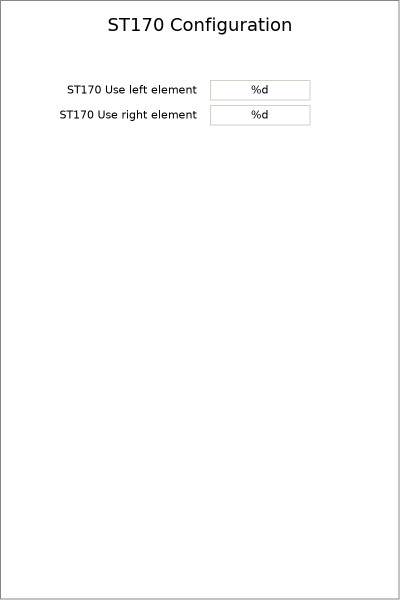
VISUALIZATION VISU_Recipe_ST170  // 400x600
    Textfield (210,80 100x20), "%d", text variable: _20_AUTO.recipe.st170.Use_element_left
        OnMouseDown: write the text variable via Default
    Label (0,5 400x40), "ST170 Configuration"
    Label (0,80 200x20), "ST170 Use left element"
    Textfield (210,105 100x20), "%d", text variable: _20_AUTO.recipe.st170.Use_element_right
        OnMouseDown: write the text variable via Default
    Label (0,105 200x20), "ST170 Use right element"
END_VISUALIZATION

(* stored: Version 1.1.0.1, ProductVersion 3.1.4024.6
   Visu VISU_Recipe_ST170: Id {58aa6de9-88ae-4e12-819a-701cfe6eed74} *)
